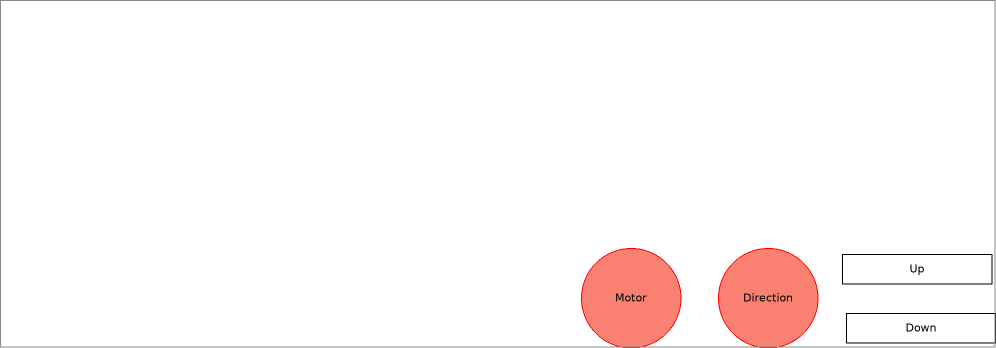
VISUALIZATION Visualization  // 996x348
    Rectangle (842,254 150x30), "Up"
        OnMouseDown: toggle POU.upButton
        OnMouseUp: toggle POU.upButton
    Rectangle (846,313 150x30), "Down"
        OnMouseDown: toggle POU.downButton
        OnMouseUp: toggle POU.downButton
    Ellipse (718,248 100x100), "Direction", colour toggle: POU.direction
    Ellipse (581,248 100x100), "Motor", colour toggle: POU.run
END_VISUALIZATION

(* stored: Version 1.1.0.1, ProductVersion 3.1.4024.3
   Visu Visualization: Id {d94e6983-ea92-48bd-9ca8-658ef0fdabcc} *)
